// TIA Portal V14 export
// export: Created 2017-01-12T07:59:05.527408Z, ExportSetting None, DisplayName Totally Integrated Automation Portal, DisplayVersion V14, DisplayName TIA Portal Openness, DisplayVersion V14, DisplayName TIA Portal Teamcenter Gateway, DisplayVersion V14, DisplayName SINAMICS Startdrive, DisplayVersion V14, DisplayName STEP 7 Professional, DisplayVersion V14, DisplayName STEP 7 Safety, DisplayVersion V14, DisplayName WinCC Advanced, DisplayVersion V14
DATA_BLOCK "General VSV"   // DB14
TITLE = VSV algemeen
{ S7_Optimized_Access := 'TRUE' }
VERSION : 3.4
// stored: AutoNumber false, MemoryReserve 100
   VAR RETAIN
      alarm : Bool;
      warning : Bool;
      Zone : Array[0..255] of Struct
         alarm : Bool;
         warning : Bool;
         lamp : Bool;
         klaxon : Bool;
         reset : Bool;
         resetklaxon : Bool;
      END_STRUCT;
   END_VAR
BEGIN
END_DATA_BLOCK
